// TIA Portal V20 export
// export: Created 2026-09-14T14:23:31.3358978Z, ExportSetting None, DisplayName Totally Integrated Automation Portal, DisplayVersion V20, DisplayName TIA Portal Openness, DisplayVersion V20, DisplayName TIA Portal Version Control Interface, DisplayVersion V20, DisplayName SINAMICS Startdrive Advanced, DisplayVersion V20, DisplayName SINAMICS Startdrive G130, G150, S120, S150, SINAMICS MV, G220, S200, S210, DisplayVersion V20, DisplayName SINAMICS Startdrive G110M, G120, G120C, G120D, G120P, G115D, DisplayVersion V20, DisplayName STEP 7 Professional, DisplayVersion V20, DisplayName STEP 7 Safety, DisplayVersion V20, DisplayName WinCC Basic/Comfort/Advanced, DisplayVersion V20, DisplayName WinCC Unified, DisplayVersion V20
ORGANIZATION_BLOCK "Main"   // OB1, LAD, ProgramCycle
TITLE = "Main Program Sweep (Cycle)"
{ S7_Optimized_Access := 'TRUE' }
// stored: AutoNumber false, SetENOAutomatically false
   VAR_INPUT
      Initial_Call : Bool;
      Remanence : Bool;
   END_VAR
BEGIN

REGION Network 1: 起保停自锁
   // 急停 %I0.2(常闭) 与 停止按钮 %I0.1 串联；启动 %I0.0 与自保持触点 %M0.0 并联后驱动运行标志
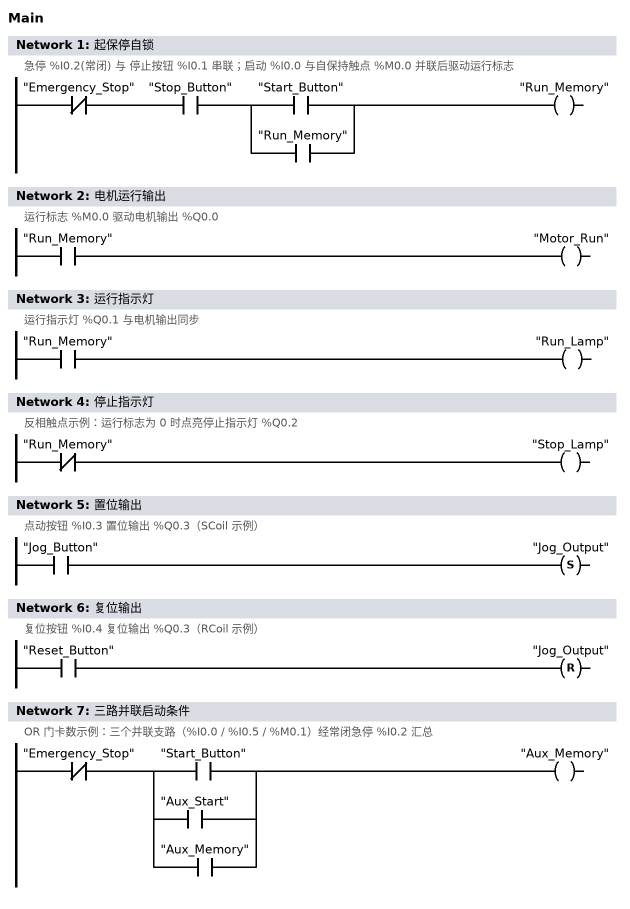
   RUNG wire#powerrail
      I_Contact( "Emergency_Stop" )
      Contact( "Stop_Button" )
      wire#w1
      Contact( "Start_Button" )
      wire#w2
      Coil( "Run_Memory" )
   END_RUNG
   RUNG wire#w1
      Contact( "Run_Memory" )
   END_RUNG wire#w2
   // the same network as SCL:
   "Run_Memory" := NOT "Emergency_Stop" AND "Stop_Button" AND ("Start_Button" OR "Run_Memory");
END_REGION

REGION Network 2: 电机运行输出
   // 运行标志 %M0.0 驱动电机输出 %Q0.0
   RUNG wire#powerrail
      Contact( "Run_Memory" )
      Coil( "Motor_Run" )
   END_RUNG
   // the same network as SCL:
   "Motor_Run" := "Run_Memory";
END_REGION

REGION Network 3: 运行指示灯
   // 运行指示灯 %Q0.1 与电机输出同步
   RUNG wire#powerrail
      Contact( "Run_Memory" )
      Coil( "Run_Lamp" )
   END_RUNG
   // the same network as SCL:
   "Run_Lamp" := "Run_Memory";
END_REGION

REGION Network 4: 停止指示灯
   // 反相触点示例：运行标志为 0 时点亮停止指示灯 %Q0.2
   RUNG wire#powerrail
      I_Contact( "Run_Memory" )
      Coil( "Stop_Lamp" )
   END_RUNG
   // the same network as SCL:
   "Stop_Lamp" := NOT "Run_Memory";
END_REGION

REGION Network 5: 置位输出
   // 点动按钮 %I0.3 置位输出 %Q0.3（SCoil 示例）
   RUNG wire#powerrail
      Contact( "Jog_Button" )
      S_Coil( "Jog_Output" )
   END_RUNG
   // the same network as SCL:
   IF "Jog_Button" THEN "Jog_Output" := TRUE; END_IF;
END_REGION

REGION Network 6: 复位输出
   // 复位按钮 %I0.4 复位输出 %Q0.3（RCoil 示例）
   RUNG wire#powerrail
      Contact( "Reset_Button" )
      R_Coil( "Jog_Output" )
   END_RUNG
   // the same network as SCL:
   IF "Reset_Button" THEN "Jog_Output" := FALSE; END_IF;
END_REGION

REGION Network 7: 三路并联启动条件
   // OR 门卡数示例：三个并联支路（%I0.0 / %I0.5 / %M0.1）经常闭急停 %I0.2 汇总
   RUNG wire#powerrail
      I_Contact( "Emergency_Stop" )
      wire#w1
      Contact( "Start_Button" )
      wire#w2
      Coil( "Aux_Memory" )
   END_RUNG
   RUNG wire#w1
      Contact( "Aux_Start" )
   END_RUNG wire#w2
   RUNG wire#w1
      Contact( "Aux_Memory" )
   END_RUNG wire#w2
   // the same network as SCL:
   "Aux_Memory" := NOT "Emergency_Stop" AND ("Start_Button" OR "Aux_Start" OR "Aux_Memory");
END_REGION
END_ORGANIZATION_BLOCK
